Fanuc KAREL source: kt00718.KL

-- PROVISIONAL review KL for V1013-1; original PC SHA256 3f139206c568b73c3de3be9c07344388d9b1b0068d55d0b33f8799a863110946
-- Incomplete behavior may be omitted. Consult companion uncertainty JSON. Do not deploy.
PROGRAM KT00718
%NOLOCKGROUP
VAR
  OUT : BOOLEAN
-- UNRESOLVED_DECL P1 type=000101
-- UNRESOLVED_DECL P2 type=000101
BEGIN
  -- UNRESOLVED_PC offsets 5-20; opcodes 22,63,23
  -- UNRESOLVED_PC offsets 25-29; opcodes 7F
END KT00718
